FUNCTION_BLOCK IA_Lighting (* ISOBUS Adapter for Lighting Data (LD) *)
  (* Standard: ISO 11783-7; Classification: PGN 65088; Description: Copyright (c) 2024-2026 HR Agrartechnik GmbH This program and the accompanying materials are made available under the terms of the Eclipse Public License 2.0 which is available at https://www.eclipse.org/legal/epl-2.0/ SPDX-License-Identifier: EPL-2.0 *)
  (* Version 1.0, 2026-04-24, Franz Höpfinger, HR Agrartechnik GmbH, initial API and implementation (Adapter Wrapper for I_Lighting) *)
  PACKAGE isobus::tecu;
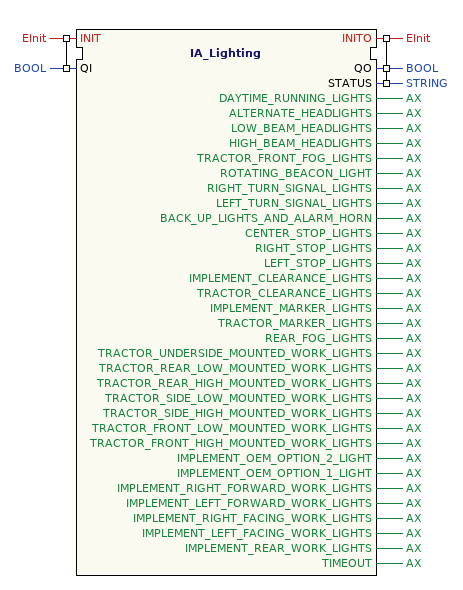
  EVENT_INPUT
    INIT : EInit WITH QI; (* Service Initialization *)
  END_EVENT
  EVENT_OUTPUT
    INITO : EInit WITH QO, STATUS; (* Initialization Confirm *)
  END_EVENT
  VAR_INPUT
    QI : BOOL; (* Event Input Qualifier *)
  END_VAR
  VAR_OUTPUT
    QO : BOOL; (* Event Output Qualifier *)
    STATUS : STRING;
  END_VAR
  PLUGS
    DAYTIME_RUNNING_LIGHTS : adapter::types::unidirectional::AX; (* Daytime Running Lights *)
    ALTERNATE_HEADLIGHTS : adapter::types::unidirectional::AX; (* Alternate Headlights *)
    LOW_BEAM_HEADLIGHTS : adapter::types::unidirectional::AX; (* Low Beam Headlights *)
    HIGH_BEAM_HEADLIGHTS : adapter::types::unidirectional::AX; (* High Beam Headlights *)
    TRACTOR_FRONT_FOG_LIGHTS : adapter::types::unidirectional::AX; (* Tractor Front Fog Lights *)
    ROTATING_BEACON_LIGHT : adapter::types::unidirectional::AX; (* Rotating Beacon Light *)
    RIGHT_TURN_SIGNAL_LIGHTS : adapter::types::unidirectional::AX; (* Right Turn Signal Lights *)
    LEFT_TURN_SIGNAL_LIGHTS : adapter::types::unidirectional::AX; (* Left Turn Signal Lights *)
    BACK_UP_LIGHTS_AND_ALARM_HORN : adapter::types::unidirectional::AX; (* Back Up Lights And Alarm Horn *)
    CENTER_STOP_LIGHTS : adapter::types::unidirectional::AX; (* Center Stop Lights *)
    RIGHT_STOP_LIGHTS : adapter::types::unidirectional::AX; (* Right Stop Lights *)
    LEFT_STOP_LIGHTS : adapter::types::unidirectional::AX; (* Left Stop Lights *)
    IMPLEMENT_CLEARANCE_LIGHTS : adapter::types::unidirectional::AX; (* Implement Clearance Lights *)
    TRACTOR_CLEARANCE_LIGHTS : adapter::types::unidirectional::AX; (* Tractor Clearance Lights *)
    IMPLEMENT_MARKER_LIGHTS : adapter::types::unidirectional::AX; (* Implement Marker Lights *)
    TRACTOR_MARKER_LIGHTS : adapter::types::unidirectional::AX; (* Tractor Marker Lights *)
    REAR_FOG_LIGHTS : adapter::types::unidirectional::AX; (* Rear Fog Lights *)
    TRACTOR_UNDERSIDE_MOUNTED_WORK_LIGHTS : adapter::types::unidirectional::AX; (* Tractor Underside Mounted Work Lights *)
    TRACTOR_REAR_LOW_MOUNTED_WORK_LIGHTS : adapter::types::unidirectional::AX; (* Tractor Rear Low Mounted Work Lights *)
    TRACTOR_REAR_HIGH_MOUNTED_WORK_LIGHTS : adapter::types::unidirectional::AX; (* Tractor Rear High Mounted Work Lights *)
    TRACTOR_SIDE_LOW_MOUNTED_WORK_LIGHTS : adapter::types::unidirectional::AX; (* Tractor Side Low Mounted Work Lights *)
    TRACTOR_SIDE_HIGH_MOUNTED_WORK_LIGHTS : adapter::types::unidirectional::AX; (* Tractor Side High Mounted Work Lights *)
    TRACTOR_FRONT_LOW_MOUNTED_WORK_LIGHTS : adapter::types::unidirectional::AX; (* Tractor Front Low Mounted Work Lights *)
    TRACTOR_FRONT_HIGH_MOUNTED_WORK_LIGHTS : adapter::types::unidirectional::AX; (* Tractor Front High Mounted Work Lights *)
    IMPLEMENT_OEM_OPTION_2_LIGHT : adapter::types::unidirectional::AX; (* Implement Oem Option 2 Light *)
    IMPLEMENT_OEM_OPTION_1_LIGHT : adapter::types::unidirectional::AX; (* Implement Oem Option 1 Light *)
    IMPLEMENT_RIGHT_FORWARD_WORK_LIGHTS : adapter::types::unidirectional::AX; (* Implement Right Forward Work Lights *)
    IMPLEMENT_LEFT_FORWARD_WORK_LIGHTS : adapter::types::unidirectional::AX; (* Implement Left Forward Work Lights *)
    IMPLEMENT_RIGHT_FACING_WORK_LIGHTS : adapter::types::unidirectional::AX; (* Implement Right Facing Work Lights *)
    IMPLEMENT_LEFT_FACING_WORK_LIGHTS : adapter::types::unidirectional::AX; (* Implement Left Facing Work Lights *)
    IMPLEMENT_REAR_WORK_LIGHTS : adapter::types::unidirectional::AX; (* Implement Rear Work Lights *)
    TIMEOUT : adapter::types::unidirectional::AX; (* Timeout Status *)
  END_PLUGS
  FBS
    I_CORE : isobus::tecu::I_Lighting;
    C_DAYTIME_RUNNING_LIGHTS : logiBUS::utils::quarter::QUARTER_TO_BOOL;
    C_ALTERNATE_HEADLIGHTS : logiBUS::utils::quarter::QUARTER_TO_BOOL;
    C_LOW_BEAM_HEADLIGHTS : logiBUS::utils::quarter::QUARTER_TO_BOOL;
    C_HIGH_BEAM_HEADLIGHTS : logiBUS::utils::quarter::QUARTER_TO_BOOL;
    C_TRACTOR_FRONT_FOG_LIGHTS : logiBUS::utils::quarter::QUARTER_TO_BOOL;
    C_ROTATING_BEACON_LIGHT : logiBUS::utils::quarter::QUARTER_TO_BOOL;
    C_RIGHT_TURN_SIGNAL_LIGHTS : logiBUS::utils::quarter::QUARTER_TO_BOOL;
    C_LEFT_TURN_SIGNAL_LIGHTS : logiBUS::utils::quarter::QUARTER_TO_BOOL;
    C_BACK_UP_LIGHTS_AND_ALARM_HORN : logiBUS::utils::quarter::QUARTER_TO_BOOL;
    C_CENTER_STOP_LIGHTS : logiBUS::utils::quarter::QUARTER_TO_BOOL;
    C_RIGHT_STOP_LIGHTS : logiBUS::utils::quarter::QUARTER_TO_BOOL;
    C_LEFT_STOP_LIGHTS : logiBUS::utils::quarter::QUARTER_TO_BOOL;
    C_IMPLEMENT_CLEARANCE_LIGHTS : logiBUS::utils::quarter::QUARTER_TO_BOOL;
    C_TRACTOR_CLEARANCE_LIGHTS : logiBUS::utils::quarter::QUARTER_TO_BOOL;
    C_IMPLEMENT_MARKER_LIGHTS : logiBUS::utils::quarter::QUARTER_TO_BOOL;
    C_TRACTOR_MARKER_LIGHTS : logiBUS::utils::quarter::QUARTER_TO_BOOL;
    C_REAR_FOG_LIGHTS : logiBUS::utils::quarter::QUARTER_TO_BOOL;
    C_TRACTOR_UNDERSIDE_MOUNTED_WORK_LIGHTS : logiBUS::utils::quarter::QUARTER_TO_BOOL;
    C_TRACTOR_REAR_LOW_MOUNTED_WORK_LIGHTS : logiBUS::utils::quarter::QUARTER_TO_BOOL;
    C_TRACTOR_REAR_HIGH_MOUNTED_WORK_LIGHTS : logiBUS::utils::quarter::QUARTER_TO_BOOL;
    C_TRACTOR_SIDE_LOW_MOUNTED_WORK_LIGHTS : logiBUS::utils::quarter::QUARTER_TO_BOOL;
    C_TRACTOR_SIDE_HIGH_MOUNTED_WORK_LIGHTS : logiBUS::utils::quarter::QUARTER_TO_BOOL;
    C_TRACTOR_FRONT_LOW_MOUNTED_WORK_LIGHTS : logiBUS::utils::quarter::QUARTER_TO_BOOL;
    C_TRACTOR_FRONT_HIGH_MOUNTED_WORK_LIGHTS : logiBUS::utils::quarter::QUARTER_TO_BOOL;
    C_IMPLEMENT_OEM_OPTION_2_LIGHT : logiBUS::utils::quarter::QUARTER_TO_BOOL;
    C_IMPLEMENT_OEM_OPTION_1_LIGHT : logiBUS::utils::quarter::QUARTER_TO_BOOL;
    C_IMPLEMENT_RIGHT_FORWARD_WORK_LIGHTS : logiBUS::utils::quarter::QUARTER_TO_BOOL;
    C_IMPLEMENT_LEFT_FORWARD_WORK_LIGHTS : logiBUS::utils::quarter::QUARTER_TO_BOOL;
    C_IMPLEMENT_RIGHT_FACING_WORK_LIGHTS : logiBUS::utils::quarter::QUARTER_TO_BOOL;
    C_IMPLEMENT_LEFT_FACING_WORK_LIGHTS : logiBUS::utils::quarter::QUARTER_TO_BOOL;
    C_IMPLEMENT_REAR_WORK_LIGHTS : logiBUS::utils::quarter::QUARTER_TO_BOOL;
  END_FBS
  EVENT_CONNECTIONS
    INIT TO I_CORE.INIT;
    I_CORE.INITO TO INITO;
    I_CORE.IND TO C_DAYTIME_RUNNING_LIGHTS.REQ;
    C_DAYTIME_RUNNING_LIGHTS.CNF TO DAYTIME_RUNNING_LIGHTS.E1;
    I_CORE.IND TO C_ALTERNATE_HEADLIGHTS.REQ;
    C_ALTERNATE_HEADLIGHTS.CNF TO ALTERNATE_HEADLIGHTS.E1;
    I_CORE.IND TO C_LOW_BEAM_HEADLIGHTS.REQ;
    C_LOW_BEAM_HEADLIGHTS.CNF TO LOW_BEAM_HEADLIGHTS.E1;
    I_CORE.IND TO C_HIGH_BEAM_HEADLIGHTS.REQ;
    C_HIGH_BEAM_HEADLIGHTS.CNF TO HIGH_BEAM_HEADLIGHTS.E1;
    I_CORE.IND TO C_TRACTOR_FRONT_FOG_LIGHTS.REQ;
    C_TRACTOR_FRONT_FOG_LIGHTS.CNF TO TRACTOR_FRONT_FOG_LIGHTS.E1;
    I_CORE.IND TO C_ROTATING_BEACON_LIGHT.REQ;
    C_ROTATING_BEACON_LIGHT.CNF TO ROTATING_BEACON_LIGHT.E1;
    I_CORE.IND TO C_RIGHT_TURN_SIGNAL_LIGHTS.REQ;
    C_RIGHT_TURN_SIGNAL_LIGHTS.CNF TO RIGHT_TURN_SIGNAL_LIGHTS.E1;
    I_CORE.IND TO C_LEFT_TURN_SIGNAL_LIGHTS.REQ;
    C_LEFT_TURN_SIGNAL_LIGHTS.CNF TO LEFT_TURN_SIGNAL_LIGHTS.E1;
    I_CORE.IND TO C_BACK_UP_LIGHTS_AND_ALARM_HORN.REQ;
    C_BACK_UP_LIGHTS_AND_ALARM_HORN.CNF TO BACK_UP_LIGHTS_AND_ALARM_HORN.E1;
    I_CORE.IND TO C_CENTER_STOP_LIGHTS.REQ;
    C_CENTER_STOP_LIGHTS.CNF TO CENTER_STOP_LIGHTS.E1;
    I_CORE.IND TO C_RIGHT_STOP_LIGHTS.REQ;
    C_RIGHT_STOP_LIGHTS.CNF TO RIGHT_STOP_LIGHTS.E1;
    I_CORE.IND TO C_LEFT_STOP_LIGHTS.REQ;
    C_LEFT_STOP_LIGHTS.CNF TO LEFT_STOP_LIGHTS.E1;
    I_CORE.IND TO C_IMPLEMENT_CLEARANCE_LIGHTS.REQ;
    C_IMPLEMENT_CLEARANCE_LIGHTS.CNF TO IMPLEMENT_CLEARANCE_LIGHTS.E1;
    I_CORE.IND TO C_TRACTOR_CLEARANCE_LIGHTS.REQ;
    C_TRACTOR_CLEARANCE_LIGHTS.CNF TO TRACTOR_CLEARANCE_LIGHTS.E1;
    I_CORE.IND TO C_IMPLEMENT_MARKER_LIGHTS.REQ;
    C_IMPLEMENT_MARKER_LIGHTS.CNF TO IMPLEMENT_MARKER_LIGHTS.E1;
    I_CORE.IND TO C_TRACTOR_MARKER_LIGHTS.REQ;
    C_TRACTOR_MARKER_LIGHTS.CNF TO TRACTOR_MARKER_LIGHTS.E1;
    I_CORE.IND TO C_REAR_FOG_LIGHTS.REQ;
    C_REAR_FOG_LIGHTS.CNF TO REAR_FOG_LIGHTS.E1;
    I_CORE.IND TO C_TRACTOR_UNDERSIDE_MOUNTED_WORK_LIGHTS.REQ;
    C_TRACTOR_UNDERSIDE_MOUNTED_WORK_LIGHTS.CNF TO TRACTOR_UNDERSIDE_MOUNTED_WORK_LIGHTS.E1;
    I_CORE.IND TO C_TRACTOR_REAR_LOW_MOUNTED_WORK_LIGHTS.REQ;
    C_TRACTOR_REAR_LOW_MOUNTED_WORK_LIGHTS.CNF TO TRACTOR_REAR_LOW_MOUNTED_WORK_LIGHTS.E1;
    I_CORE.IND TO C_TRACTOR_REAR_HIGH_MOUNTED_WORK_LIGHTS.REQ;
    C_TRACTOR_REAR_HIGH_MOUNTED_WORK_LIGHTS.CNF TO TRACTOR_REAR_HIGH_MOUNTED_WORK_LIGHTS.E1;
    I_CORE.IND TO C_TRACTOR_SIDE_LOW_MOUNTED_WORK_LIGHTS.REQ;
    C_TRACTOR_SIDE_LOW_MOUNTED_WORK_LIGHTS.CNF TO TRACTOR_SIDE_LOW_MOUNTED_WORK_LIGHTS.E1;
    I_CORE.IND TO C_TRACTOR_SIDE_HIGH_MOUNTED_WORK_LIGHTS.REQ;
    C_TRACTOR_SIDE_HIGH_MOUNTED_WORK_LIGHTS.CNF TO TRACTOR_SIDE_HIGH_MOUNTED_WORK_LIGHTS.E1;
    I_CORE.IND TO C_TRACTOR_FRONT_LOW_MOUNTED_WORK_LIGHTS.REQ;
    C_TRACTOR_FRONT_LOW_MOUNTED_WORK_LIGHTS.CNF TO TRACTOR_FRONT_LOW_MOUNTED_WORK_LIGHTS.E1;
    I_CORE.IND TO C_TRACTOR_FRONT_HIGH_MOUNTED_WORK_LIGHTS.REQ;
    C_TRACTOR_FRONT_HIGH_MOUNTED_WORK_LIGHTS.CNF TO TRACTOR_FRONT_HIGH_MOUNTED_WORK_LIGHTS.E1;
    I_CORE.IND TO C_IMPLEMENT_OEM_OPTION_2_LIGHT.REQ;
    C_IMPLEMENT_OEM_OPTION_2_LIGHT.CNF TO IMPLEMENT_OEM_OPTION_2_LIGHT.E1;
    I_CORE.IND TO C_IMPLEMENT_OEM_OPTION_1_LIGHT.REQ;
    C_IMPLEMENT_OEM_OPTION_1_LIGHT.CNF TO IMPLEMENT_OEM_OPTION_1_LIGHT.E1;
    I_CORE.IND TO C_IMPLEMENT_RIGHT_FORWARD_WORK_LIGHTS.REQ;
    C_IMPLEMENT_RIGHT_FORWARD_WORK_LIGHTS.CNF TO IMPLEMENT_RIGHT_FORWARD_WORK_LIGHTS.E1;
    I_CORE.IND TO C_IMPLEMENT_LEFT_FORWARD_WORK_LIGHTS.REQ;
    C_IMPLEMENT_LEFT_FORWARD_WORK_LIGHTS.CNF TO IMPLEMENT_LEFT_FORWARD_WORK_LIGHTS.E1;
    I_CORE.IND TO C_IMPLEMENT_RIGHT_FACING_WORK_LIGHTS.REQ;
    C_IMPLEMENT_RIGHT_FACING_WORK_LIGHTS.CNF TO IMPLEMENT_RIGHT_FACING_WORK_LIGHTS.E1;
    I_CORE.IND TO C_IMPLEMENT_LEFT_FACING_WORK_LIGHTS.REQ;
    C_IMPLEMENT_LEFT_FACING_WORK_LIGHTS.CNF TO IMPLEMENT_LEFT_FACING_WORK_LIGHTS.E1;
    I_CORE.IND TO C_IMPLEMENT_REAR_WORK_LIGHTS.REQ;
    C_IMPLEMENT_REAR_WORK_LIGHTS.CNF TO IMPLEMENT_REAR_WORK_LIGHTS.E1;
    I_CORE.TIMEOUT TO TIMEOUT.E1;
  END_CONNECTIONS
  DATA_CONNECTIONS
    QI TO I_CORE.QI;
    I_CORE.QO TO QO;
    I_CORE.STATUS TO STATUS;
    I_CORE.DAYTIME_RUNNING_LIGHTS TO C_DAYTIME_RUNNING_LIGHTS.IB;
    C_DAYTIME_RUNNING_LIGHTS.Q TO DAYTIME_RUNNING_LIGHTS.D1;
    I_CORE.ALTERNATE_HEADLIGHTS TO C_ALTERNATE_HEADLIGHTS.IB;
    C_ALTERNATE_HEADLIGHTS.Q TO ALTERNATE_HEADLIGHTS.D1;
    I_CORE.LOW_BEAM_HEADLIGHTS TO C_LOW_BEAM_HEADLIGHTS.IB;
    C_LOW_BEAM_HEADLIGHTS.Q TO LOW_BEAM_HEADLIGHTS.D1;
    I_CORE.HIGH_BEAM_HEADLIGHTS TO C_HIGH_BEAM_HEADLIGHTS.IB;
    C_HIGH_BEAM_HEADLIGHTS.Q TO HIGH_BEAM_HEADLIGHTS.D1;
    I_CORE.TRACTOR_FRONT_FOG_LIGHTS TO C_TRACTOR_FRONT_FOG_LIGHTS.IB;
    C_TRACTOR_FRONT_FOG_LIGHTS.Q TO TRACTOR_FRONT_FOG_LIGHTS.D1;
    I_CORE.ROTATING_BEACON_LIGHT TO C_ROTATING_BEACON_LIGHT.IB;
    C_ROTATING_BEACON_LIGHT.Q TO ROTATING_BEACON_LIGHT.D1;
    I_CORE.RIGHT_TURN_SIGNAL_LIGHTS TO C_RIGHT_TURN_SIGNAL_LIGHTS.IB;
    C_RIGHT_TURN_SIGNAL_LIGHTS.Q TO RIGHT_TURN_SIGNAL_LIGHTS.D1;
    I_CORE.LEFT_TURN_SIGNAL_LIGHTS TO C_LEFT_TURN_SIGNAL_LIGHTS.IB;
    C_LEFT_TURN_SIGNAL_LIGHTS.Q TO LEFT_TURN_SIGNAL_LIGHTS.D1;
    I_CORE.BACK_UP_LIGHTS_AND_ALARM_HORN TO C_BACK_UP_LIGHTS_AND_ALARM_HORN.IB;
    C_BACK_UP_LIGHTS_AND_ALARM_HORN.Q TO BACK_UP_LIGHTS_AND_ALARM_HORN.D1;
    I_CORE.CENTER_STOP_LIGHTS TO C_CENTER_STOP_LIGHTS.IB;
    C_CENTER_STOP_LIGHTS.Q TO CENTER_STOP_LIGHTS.D1;
    I_CORE.RIGHT_STOP_LIGHTS TO C_RIGHT_STOP_LIGHTS.IB;
    C_RIGHT_STOP_LIGHTS.Q TO RIGHT_STOP_LIGHTS.D1;
    I_CORE.LEFT_STOP_LIGHTS TO C_LEFT_STOP_LIGHTS.IB;
    C_LEFT_STOP_LIGHTS.Q TO LEFT_STOP_LIGHTS.D1;
    I_CORE.IMPLEMENT_CLEARANCE_LIGHTS TO C_IMPLEMENT_CLEARANCE_LIGHTS.IB;
    C_IMPLEMENT_CLEARANCE_LIGHTS.Q TO IMPLEMENT_CLEARANCE_LIGHTS.D1;
    I_CORE.TRACTOR_CLEARANCE_LIGHTS TO C_TRACTOR_CLEARANCE_LIGHTS.IB;
    C_TRACTOR_CLEARANCE_LIGHTS.Q TO TRACTOR_CLEARANCE_LIGHTS.D1;
    I_CORE.IMPLEMENT_MARKER_LIGHTS TO C_IMPLEMENT_MARKER_LIGHTS.IB;
    C_IMPLEMENT_MARKER_LIGHTS.Q TO IMPLEMENT_MARKER_LIGHTS.D1;
    I_CORE.TRACTOR_MARKER_LIGHTS TO C_TRACTOR_MARKER_LIGHTS.IB;
    C_TRACTOR_MARKER_LIGHTS.Q TO TRACTOR_MARKER_LIGHTS.D1;
    I_CORE.REAR_FOG_LIGHTS TO C_REAR_FOG_LIGHTS.IB;
    C_REAR_FOG_LIGHTS.Q TO REAR_FOG_LIGHTS.D1;
    I_CORE.TRACTOR_UNDERSIDE_MOUNTED_WORK_LIGHTS TO C_TRACTOR_UNDERSIDE_MOUNTED_WORK_LIGHTS.IB;
    C_TRACTOR_UNDERSIDE_MOUNTED_WORK_LIGHTS.Q TO TRACTOR_UNDERSIDE_MOUNTED_WORK_LIGHTS.D1;
    I_CORE.TRACTOR_REAR_LOW_MOUNTED_WORK_LIGHTS TO C_TRACTOR_REAR_LOW_MOUNTED_WORK_LIGHTS.IB;
    C_TRACTOR_REAR_LOW_MOUNTED_WORK_LIGHTS.Q TO TRACTOR_REAR_LOW_MOUNTED_WORK_LIGHTS.D1;
    I_CORE.TRACTOR_REAR_HIGH_MOUNTED_WORK_LIGHTS TO C_TRACTOR_REAR_HIGH_MOUNTED_WORK_LIGHTS.IB;
    C_TRACTOR_REAR_HIGH_MOUNTED_WORK_LIGHTS.Q TO TRACTOR_REAR_HIGH_MOUNTED_WORK_LIGHTS.D1;
    I_CORE.TRACTOR_SIDE_LOW_MOUNTED_WORK_LIGHTS TO C_TRACTOR_SIDE_LOW_MOUNTED_WORK_LIGHTS.IB;
    C_TRACTOR_SIDE_LOW_MOUNTED_WORK_LIGHTS.Q TO TRACTOR_SIDE_LOW_MOUNTED_WORK_LIGHTS.D1;
    I_CORE.TRACTOR_SIDE_HIGH_MOUNTED_WORK_LIGHTS TO C_TRACTOR_SIDE_HIGH_MOUNTED_WORK_LIGHTS.IB;
    C_TRACTOR_SIDE_HIGH_MOUNTED_WORK_LIGHTS.Q TO TRACTOR_SIDE_HIGH_MOUNTED_WORK_LIGHTS.D1;
    I_CORE.TRACTOR_FRONT_LOW_MOUNTED_WORK_LIGHTS TO C_TRACTOR_FRONT_LOW_MOUNTED_WORK_LIGHTS.IB;
    C_TRACTOR_FRONT_LOW_MOUNTED_WORK_LIGHTS.Q TO TRACTOR_FRONT_LOW_MOUNTED_WORK_LIGHTS.D1;
    I_CORE.TRACTOR_FRONT_HIGH_MOUNTED_WORK_LIGHTS TO C_TRACTOR_FRONT_HIGH_MOUNTED_WORK_LIGHTS.IB;
    C_TRACTOR_FRONT_HIGH_MOUNTED_WORK_LIGHTS.Q TO TRACTOR_FRONT_HIGH_MOUNTED_WORK_LIGHTS.D1;
    I_CORE.IMPLEMENT_OEM_OPTION_2_LIGHT TO C_IMPLEMENT_OEM_OPTION_2_LIGHT.IB;
    C_IMPLEMENT_OEM_OPTION_2_LIGHT.Q TO IMPLEMENT_OEM_OPTION_2_LIGHT.D1;
    I_CORE.IMPLEMENT_OEM_OPTION_1_LIGHT TO C_IMPLEMENT_OEM_OPTION_1_LIGHT.IB;
    C_IMPLEMENT_OEM_OPTION_1_LIGHT.Q TO IMPLEMENT_OEM_OPTION_1_LIGHT.D1;
    I_CORE.IMPLEMENT_RIGHT_FORWARD_WORK_LIGHTS TO C_IMPLEMENT_RIGHT_FORWARD_WORK_LIGHTS.IB;
    C_IMPLEMENT_RIGHT_FORWARD_WORK_LIGHTS.Q TO IMPLEMENT_RIGHT_FORWARD_WORK_LIGHTS.D1;
    I_CORE.IMPLEMENT_LEFT_FORWARD_WORK_LIGHTS TO C_IMPLEMENT_LEFT_FORWARD_WORK_LIGHTS.IB;
    C_IMPLEMENT_LEFT_FORWARD_WORK_LIGHTS.Q TO IMPLEMENT_LEFT_FORWARD_WORK_LIGHTS.D1;
    I_CORE.IMPLEMENT_RIGHT_FACING_WORK_LIGHTS TO C_IMPLEMENT_RIGHT_FACING_WORK_LIGHTS.IB;
    C_IMPLEMENT_RIGHT_FACING_WORK_LIGHTS.Q TO IMPLEMENT_RIGHT_FACING_WORK_LIGHTS.D1;
    I_CORE.IMPLEMENT_LEFT_FACING_WORK_LIGHTS TO C_IMPLEMENT_LEFT_FACING_WORK_LIGHTS.IB;
    C_IMPLEMENT_LEFT_FACING_WORK_LIGHTS.Q TO IMPLEMENT_LEFT_FACING_WORK_LIGHTS.D1;
    I_CORE.IMPLEMENT_REAR_WORK_LIGHTS TO C_IMPLEMENT_REAR_WORK_LIGHTS.IB;
    C_IMPLEMENT_REAR_WORK_LIGHTS.Q TO IMPLEMENT_REAR_WORK_LIGHTS.D1;
    I_CORE.Q_timeout TO TIMEOUT.D1;
  END_CONNECTIONS
END_FUNCTION_BLOCK
